TYPE ST_DebugSensors_LowLiftEmulation :
STRUCT
	EnableSensorDebug	: BOOL; 					// Overwrite sensor values with debug sensor values
	HW_Inputs			: ST_HW_InputsLowLiftUnit;	// Debug sensors
END_STRUCT
END_TYPE

(* stored: Version 1.1.0.1, ProductVersion 3.1.4024.9
   DUT ST_DebugSensors_LowLiftEmulation: Id {8dc91fa1-16ba-425c-9c86-95a328abec7a} *)
